// TIA Portal V16 export
// export: Created 2021-05-26T11:52:20.6664228Z, ExportSetting WithDefaults, DisplayName Totally Integrated Automation Portal, DisplayVersion V16 Update 4, DisplayName TIA Portal Version Control Interface, DisplayVersion V16 Update 2, DisplayName TIA Portal Openness, DisplayVersion V16 Update 4, DisplayName STEP 7 Professional, DisplayVersion V16 Update 4, DisplayName STEP 7 Safety, DisplayVersion V16, DisplayName WinCC Advanced, DisplayVersion V16 Update 4
DATA_BLOCK "DB_CuVo_intAr"   // DB27
{ S7_Optimized_Access := 'FALSE'; DB_Accessible_From_OPC_UA := 'FALSE' }
VERSION : 0.1
// stored: AutoNumber true, DBAccessibleFromOPCUA false, IsOnlyStoredInLoadMemory false, IsWriteProtectedInAS false
   VAR
      swpCurM1Tr : Array[1..16] of "UDT_swp51Data";
      swpVolM1Tr { S7_SetPoint := 'True'} : Array[1..16] of "UDT_swp51Data";
      swpCurM2Tr { S7_SetPoint := 'True'} : Array[1..16] of "UDT_swp51Data";
      swpVolM2Tr { S7_SetPoint := 'True'} : Array[1..16] of "UDT_swp51Data";
      swpCurM3Tr { S7_SetPoint := 'True'} : Array[1..16] of "UDT_swp51Data";
      swpVolM3Tr { S7_SetPoint := 'True'} : Array[1..16] of "UDT_swp51Data";
      swpCurM4Tr { S7_SetPoint := 'True'} : Array[1..16] of "UDT_swp51Data";
      swpVolM4Tr { S7_SetPoint := 'True'} : Array[1..16] of "UDT_swp51Data";
      swpCurM5Tr { S7_SetPoint := 'True'} : Array[1..16] of "UDT_swp51Data";
      swpVolM5Tr { S7_SetPoint := 'True'} : Array[1..16] of "UDT_swp51Data";
      swpCurM6Tr { S7_SetPoint := 'True'} : Array[1..16] of "UDT_swp51Data";
      swpVolM6Tr { S7_SetPoint := 'True'} : Array[1..16] of "UDT_swp51Data";
      swpCurM7Tr { S7_SetPoint := 'True'} : Array[1..16] of "UDT_swp51Data";
      swpVolM7Tr { S7_SetPoint := 'True'} : Array[1..16] of "UDT_swp51Data";
      swpCurM8Tr { S7_SetPoint := 'True'} : Array[1..16] of "UDT_swp51Data";
      swpVolM8Tr { S7_SetPoint := 'True'} : Array[1..16] of "UDT_swp51Data";
      swpCurM9Tr { S7_SetPoint := 'True'} : Array[1..16] of "UDT_swp51Data";
      swpVolM9Tr { S7_SetPoint := 'True'} : Array[1..16] of "UDT_swp51Data";
      swpCurM10Tr { S7_SetPoint := 'True'} : Array[1..16] of "UDT_swp51Data";
      swpVolM10Tr { S7_SetPoint := 'True'} : Array[1..16] of "UDT_swp51Data";
      swpCurM11Tr { S7_SetPoint := 'True'} : Array[1..16] of "UDT_swp51Data";
      swpVolM11Tr { S7_SetPoint := 'True'} : Array[1..16] of "UDT_swp51Data";
      swpCurM12Tr { S7_SetPoint := 'True'} : Array[1..16] of "UDT_swp51Data";
      swpVolM12Tr { S7_SetPoint := 'True'} : Array[1..16] of "UDT_swp51Data";
      swpCurM13Tr { S7_SetPoint := 'True'} : Array[1..16] of "UDT_swp51Data";
      swpVolM13Tr { S7_SetPoint := 'True'} : Array[1..16] of "UDT_swp51Data";
      swpCurM14Tr { S7_SetPoint := 'True'} : Array[1..16] of "UDT_swp51Data";
      swpVolM14Tr { S7_SetPoint := 'True'} : Array[1..16] of "UDT_swp51Data";
      swpCurM15Tr { S7_SetPoint := 'True'} : Array[1..16] of "UDT_swp51Data";
      swpVolM15Tr { S7_SetPoint := 'True'} : Array[1..16] of "UDT_swp51Data";
   END_VAR
BEGIN
END_DATA_BLOCK
